FUNCTION_BLOCK InfoData
VAR
    {attribute addProperty Name  "<#EC State (8=OK)#>"}
    EC_State AT %I* : BOOL;
    {attribute addProperty Name  "<#EC ASM ADDR#>"}
    EC_AmsAddr AT %I* : AMSADDR;
END_VAR

END_FUNCTION_BLOCK

(* stored: Version 1.1.0.1, ProductVersion 3.1.4024.6
   POU InfoData: Id {a74f2e97-e5df-4368-bcd0-903f5fe39b86}, SpecialFunc None *)
